KUKA KRL program: ps_stb_geo_c1.src, ps_stb_geo_c1.dat

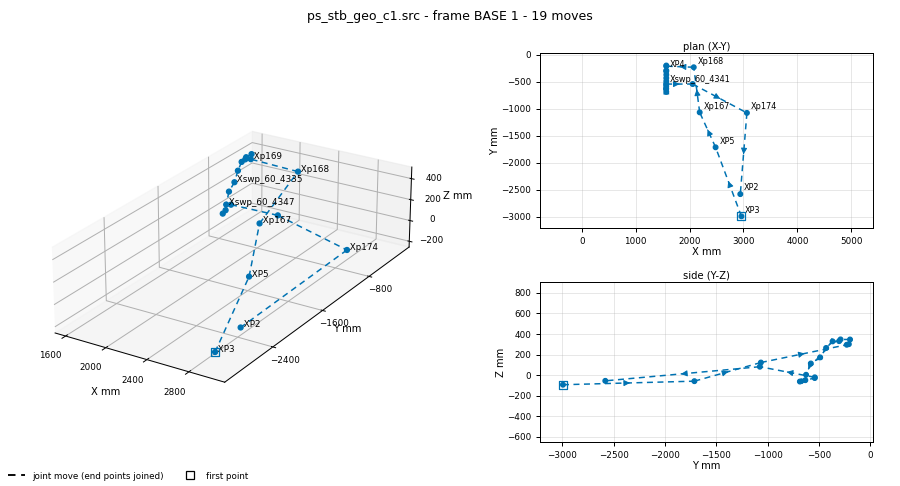
[picture p0: tool path of ps_stb_geo_c1.src in frame BASE 1, 19 of 19 moves have a stored position in this frame; points joined in program order, loops and branches not executed]
--- ps_stb_geo_c1.src ---
&ACCESS RVO
&REL 8
&COMMENT Solda GUN C1 geometria
&PARAM DISKPATH = KRC:\R1\Program
DEF ps_stb_geo_c1( )

;FOLD INI
  ;FOLD BASISTECH INI
    GLOBAL INTERRUPT DECL 3 WHEN $STOPMESS==TRUE DO IR_STOPM ( )
    INTERRUPT ON 3
    BAS (#INITMOV,0 )
  ;ENDFOLD (BASISTECH INI)
;FOLD SPOTTECH INI
USERSPOT(#INIT)
;ENDFOLD (SPOTTECH INI)
;FOLD GRIPPERTECH INI
USER_GRP(0,DUMMY,DUMMY,GDEFAULT)
;ENDFOLD (GRIPPERTECH INI)
  ;FOLD USER INI
    ;Make your modifications here

  ;ENDFOLD (USER INI)
;ENDFOLD (INI)

; Caracterização dos meios de produção:
; Versão Atual:
; 08/06/2013 12:00 Name: P13.050-R1 CHANGES: Solda geometria STB
; Gun C1 (F2 6640 0018 984)

chk_w2_wechs_ok ( )              ; CHECK C1

if MaxStandMenge (1) then
 MaxStandmengeErreicht (1)
endif

IF (NOT(GHOST())) THEN
if Elektrodenwechsel (1) then
 e_fraes2 ()
endif
ENDIF

;FOLD PTP P3 CONT Vel=100 % P_OLP23 Tool[2]:GUN C1 Base[1]:Actros;%{PE}%R 8.2.20,%MKUKATPBASIS,%CMOVE,%VPTP,%P 1:PTP, 2:P3, 3:C_DIS, 5:100, 7:P_OLP23
$BWDSTART=FALSE
PDAT_ACT=PP_OLP23
FDAT_ACT=FP3
BAS(#PTP_PARAMS,100)
PTP XP3 C_DIS
;ENDFOLD
;FOLD PTP P5 CONT Vel=100 % P_OLP24 Tool[2]:GUN C1 Base[1]:Actros;%{PE}%R 8.2.20,%MKUKATPBASIS,%CMOVE,%VPTP,%P 1:PTP, 2:P5, 3:C_DIS, 5:100, 7:P_OLP24
$BWDSTART=FALSE
PDAT_ACT=PP_OLP24
FDAT_ACT=FP5
BAS(#PTP_PARAMS,100)
PTP XP5 C_DIS
;ENDFOLD

;FOLD OUT 3339 'R1 solicita lib soldar geometria' State=TRUE ;%{PE}%R 8.2.20,%MKUKATPBASIS,%COUT,%VOUTX,%P 2:3339, 3:R1 solicita lib soldar geometria, 5:TRUE, 6:
$OUT[3339]=TRUE
;ENDFOLD
;FOLD WAIT FOR ( IN 3339 'Aguarda lib. Soldar geometria' );%{PE}%R 8.2.20,%MKUKATPBASIS,%CEXT_WAIT_FOR,%VEXT_WAIT_FOR,%P 2:, 4:, 5:$IN, 6:3339, 7:Aguarda lib. Soldar geometria, 9:
WAIT FOR  ( $IN[3339] )
;ENDFOLD
;FOLD OUT 3339 'R1 solicita lib soldar geometria' State=FALSE ;%{PE}%R 8.2.20,%MKUKATPBASIS,%COUT,%VOUTX,%P 2:3339, 3:R1 solicita lib soldar geometria, 5:FALSE, 6:
$OUT[3339]=FALSE
;ENDFOLD
;FOLD OUT 3344 'R1 entregou peça geo box' State=FALSE ;%{PE}%R 8.2.20,%MKUKATPBASIS,%COUT,%VOUTX,%P 2:3344, 3:R1 entregou peça geo box, 5:FALSE, 6:
$OUT[3344]=FALSE
;ENDFOLD
;FOLD OUT 3348 'Fora area GEOBOX' State=FALSE ;%{PE}%R 8.2.20,%MKUKATPBASIS,%COUT,%VOUTX,%P 2:3348, 3:Fora area GEOBOX, 5:FALSE, 6:
$OUT[3348]=FALSE
;ENDFOLD

;FOLD PTP p167 CONT Vel=100 % P_OLP6 Tool[2]:GUN C1 Base[1]:Actros;%{PE}%R8.2,%MKUKATPBASIS,%CMOVE,%VPTP,%P 1:PTP, 2:p167, 3:C_DIS, 5:100, 7:P_OLP6
$BWDSTART = FALSE
PDAT_ACT= PP_OLP6
FDAT_ACT= Fp167
BAS(#PTP_PARAMS,100)
PTP Xp167 C_DIS
;ENDFOLD

;FOLD Collision.Monitoring_2_On ;%{PE}%MKUKATPUSER
COLLSTOP( 2, 1 ) ;Interrupt-Controlled
;ENDFOLD

;FOLD PTP p168 CONT Vel=100 % P_OLP7 Tool[2]:GUN C1 Base[1]:Actros;%{PE}%R8.2,%MKUKATPBASIS,%CMOVE,%VPTP,%P 1:PTP, 2:p168, 3:C_DIS, 5:100, 7:P_OLP7
$BWDSTART = FALSE
PDAT_ACT= PP_OLP7
FDAT_ACT= Fp168
BAS(#PTP_PARAMS,100)
PTP Xp168 C_DIS
;ENDFOLD
;FOLD PTP p169 CONT Vel=100 % P_OLP8 Tool[2]:GUN C1 Base[1]:Actros;%{PE}%R8.2,%MKUKATPBASIS,%CMOVE,%VPTP,%P 1:PTP, 2:p169, 3:C_DIS, 5:100, 7:P_OLP8
$BWDSTART = FALSE
PDAT_ACT= PP_OLP8
FDAT_ACT= Fp169
BAS(#PTP_PARAMS,100)
PTP Xp169 C_DIS
;ENDFOLD

;FOLD ; swp_60_4311;%{PE}%R 8.2.20,%MKUKATPBASIS,%CCOMMENT,%VNORMAL,%P 2:swp_60_4311
;ENDFOLD
;FOLD PTP swp_60_4311 P_OLP9 SPOT Gun=1 RETR CLS PgNo1=38 ACTIVE=1 Tool[2]:GUN C1 Base[1]:Actros;%{PE}%R 8.2.2,%MKUKATPSPOT,%CSPOT,%VPTP,%P 1:PTP, 2:swp_60_4311, 3:, 5:100, 7:P_OLP9, 10:1, 12:#FIRST, 14:#CLO, 16:38, 18:1, 20:1, 22:0, 24:1, 25:S_OLP1
$BWDSTART=FALSE
PDAT_ACT=PP_OLP9
FDAT_ACT=Fswp_60_4311
BAS(#PTP_PARAMS,PP_OLP9.VEL)
S_ACT.GUN=1
S_ACT.PAIR=SDEFAULT.PAIR
S_ACT.RETR=#CLO
S_ACT.CLO_TM=1
S_ACT.PGNO1=38
S_ACT.PGNO2=SDEFAULT.PGNO2
S_ACT.PRESS1=SDEFAULT.PRESS1
S_ACT.PRESS2=SDEFAULT.PRESS2
S_READY=FALSE
PTP Xswp_60_4311
USERSPOT(#SPOT, S_ACT)
WAIT FOR S_READY
;ENDFOLD

;FOLD ; swp_60_4317;%{PE}%R 8.2.20,%MKUKATPBASIS,%CCOMMENT,%VNORMAL,%P 2:swp_60_4317
;ENDFOLD
;FOLD PTP swp_60_4317 P_OLP10 SPOT Gun=1 RETR CLS PgNo1=39 ACTIVE=1 Tool[2]:GUN C1 Base[1]:Actros;%{PE}%R 8.2.2,%MKUKATPSPOT,%CSPOT,%VPTP,%P 1:PTP, 2:swp_60_4317, 3:, 5:100, 7:P_OLP10, 10:1, 12:#FIRST, 14:#CLO, 16:39, 18:1, 20:1, 22:0, 24:1, 25:S_OLP2
$BWDSTART=FALSE
PDAT_ACT=PP_OLP10
FDAT_ACT=Fswp_60_4317
BAS(#PTP_PARAMS,PP_OLP10.VEL)
S_ACT.GUN=1
S_ACT.PAIR=SDEFAULT.PAIR
S_ACT.RETR=#CLO
S_ACT.CLO_TM=1
S_ACT.PGNO1=39
S_ACT.PGNO2=SDEFAULT.PGNO2
S_ACT.PRESS1=SDEFAULT.PRESS1
S_ACT.PRESS2=SDEFAULT.PRESS2
S_READY=FALSE
PTP Xswp_60_4317
USERSPOT(#SPOT, S_ACT)
WAIT FOR S_READY
;ENDFOLD

;FOLD PTP P4 CONT Vel=100 % PDAT3 Tool[2]:GUN C1 Base[1]:Actros;%{PE}%R 8.2.20,%MKUKATPBASIS,%CMOVE,%VPTP,%P 1:PTP, 2:P4, 3:C_DIS, 5:100, 7:PDAT3
$BWDSTART=FALSE
PDAT_ACT=PPDAT3
FDAT_ACT=FP4
BAS(#PTP_PARAMS,100)
PTP XP4 C_DIS
;ENDFOLD

;FOLD ; swp_60_4323;%{PE}%R 8.2.20,%MKUKATPBASIS,%CCOMMENT,%VNORMAL,%P 2:swp_60_4323
;ENDFOLD
;FOLD PTP swp_60_4323 P_OLP11 SPOT Gun=1 RETR CLS PgNo1=40 ACTIVE=1 Tool[2]:GUN C1 Base[1]:Actros;%{PE}%R 8.2.2,%MKUKATPSPOT,%CSPOT,%VPTP,%P 1:PTP, 2:swp_60_4323, 3:, 5:100, 7:P_OLP11, 10:1, 12:#FIRST, 14:#CLO, 16:40, 18:1, 20:1, 22:0, 24:1, 25:S_OLP3
$BWDSTART=FALSE
PDAT_ACT=PP_OLP11
FDAT_ACT=Fswp_60_4323
BAS(#PTP_PARAMS,PP_OLP11.VEL)
S_ACT.GUN=1
S_ACT.PAIR=SDEFAULT.PAIR
S_ACT.RETR=#CLO
S_ACT.CLO_TM=1
S_ACT.PGNO1=40
S_ACT.PGNO2=SDEFAULT.PGNO2
S_ACT.PRESS1=SDEFAULT.PRESS1
S_ACT.PRESS2=SDEFAULT.PRESS2
S_READY=FALSE
PTP Xswp_60_4323
USERSPOT(#SPOT, S_ACT)
WAIT FOR S_READY
;ENDFOLD

;FOLD ; swp_60_4329;%{PE}%R 8.2.20,%MKUKATPBASIS,%CCOMMENT,%VNORMAL,%P 2:swp_60_4329
;ENDFOLD
;FOLD PTP swp_60_4329 P_OLP12 SPOT Gun=1 RETR CLS PgNo1=41 ACTIVE=1 Tool[2]:GUN C1 Base[1]:Actros;%{PE}%R 8.2.2,%MKUKATPSPOT,%CSPOT,%VPTP,%P 1:PTP, 2:swp_60_4329, 3:, 5:100, 7:P_OLP12, 10:1, 12:#FIRST, 14:#CLO, 16:41, 18:1, 20:1, 22:0, 24:1, 25:S_OLP4
$BWDSTART=FALSE
PDAT_ACT=PP_OLP12
FDAT_ACT=Fswp_60_4329
BAS(#PTP_PARAMS,PP_OLP12.VEL)
S_ACT.GUN=1
S_ACT.PAIR=SDEFAULT.PAIR
S_ACT.RETR=#CLO
S_ACT.CLO_TM=1
S_ACT.PGNO1=41
S_ACT.PGNO2=SDEFAULT.PGNO2
S_ACT.PRESS1=SDEFAULT.PRESS1
S_ACT.PRESS2=SDEFAULT.PRESS2
S_READY=FALSE
PTP Xswp_60_4329
USERSPOT(#SPOT, S_ACT)
WAIT FOR S_READY
;ENDFOLD

;FOLD ; swp_60_4335;%{PE}%R 8.2.20,%MKUKATPBASIS,%CCOMMENT,%VNORMAL,%P 2:swp_60_4335
;ENDFOLD
;FOLD PTP swp_60_4335 P_OLP13 SPOT Gun=1 RETR CLS PgNo1=42 ACTIVE=1 Tool[2]:GUN C1 Base[1]:Actros;%{PE}%R 8.2.2,%MKUKATPSPOT,%CSPOT,%VPTP,%P 1:PTP, 2:swp_60_4335, 3:, 5:100, 7:P_OLP13, 10:1, 12:#FIRST, 14:#CLO, 16:42, 18:1, 20:1, 22:0, 24:1, 25:S_OLP5
$BWDSTART=FALSE
PDAT_ACT=PP_OLP13
FDAT_ACT=Fswp_60_4335
BAS(#PTP_PARAMS,PP_OLP13.VEL)
S_ACT.GUN=1
S_ACT.PAIR=SDEFAULT.PAIR
S_ACT.RETR=#CLO
S_ACT.CLO_TM=1
S_ACT.PGNO1=42
S_ACT.PGNO2=SDEFAULT.PGNO2
S_ACT.PRESS1=SDEFAULT.PRESS1
S_ACT.PRESS2=SDEFAULT.PRESS2
S_READY=FALSE
PTP Xswp_60_4335
USERSPOT(#SPOT, S_ACT)
WAIT FOR S_READY
;ENDFOLD

;FOLD ; swp_60_4341;%{PE}%R 8.2.20,%MKUKATPBASIS,%CCOMMENT,%VNORMAL,%P 2:swp_60_4341
;ENDFOLD
;FOLD PTP swp_60_4341 P_OLP14 SPOT Gun=1 RETR CLS PgNo1=43 ACTIVE=1 Tool[2]:GUN C1 Base[1]:Actros;%{PE}%R 8.2.2,%MKUKATPSPOT,%CSPOT,%VPTP,%P 1:PTP, 2:swp_60_4341, 3:, 5:100, 7:P_OLP14, 10:1, 12:#FIRST, 14:#CLO, 16:43, 18:1, 20:1, 22:0, 24:1, 25:S_OLP6
$BWDSTART=FALSE
PDAT_ACT=PP_OLP14
FDAT_ACT=Fswp_60_4341
BAS(#PTP_PARAMS,PP_OLP14.VEL)
S_ACT.GUN=1
S_ACT.PAIR=SDEFAULT.PAIR
S_ACT.RETR=#CLO
S_ACT.CLO_TM=1
S_ACT.PGNO1=43
S_ACT.PGNO2=SDEFAULT.PGNO2
S_ACT.PRESS1=SDEFAULT.PRESS1
S_ACT.PRESS2=SDEFAULT.PRESS2
S_READY=FALSE
PTP Xswp_60_4341
USERSPOT(#SPOT, S_ACT)
WAIT FOR S_READY
;ENDFOLD

;FOLD ; swp_60_4347;%{PE}%R 8.2.20,%MKUKATPBASIS,%CCOMMENT,%VNORMAL,%P 2:swp_60_4347
;ENDFOLD
;FOLD PTP swp_60_4347 P_OLP15 SPOT Gun=1 RETR CLS PgNo1=44 ACTIVE=1 Tool[2]:GUN C1 Base[1]:Actros;%{PE}%R 8.2.2,%MKUKATPSPOT,%CSPOT,%VPTP,%P 1:PTP, 2:swp_60_4347, 3:, 5:100, 7:P_OLP15, 10:1, 12:#FIRST, 14:#CLO, 16:44, 18:1, 20:1, 22:0, 24:1, 25:S_OLP7
$BWDSTART=FALSE
PDAT_ACT=PP_OLP15
FDAT_ACT=Fswp_60_4347
BAS(#PTP_PARAMS,PP_OLP15.VEL)
S_ACT.GUN=1
S_ACT.PAIR=SDEFAULT.PAIR
S_ACT.RETR=#CLO
S_ACT.CLO_TM=1
S_ACT.PGNO1=44
S_ACT.PGNO2=SDEFAULT.PGNO2
S_ACT.PRESS1=SDEFAULT.PRESS1
S_ACT.PRESS2=SDEFAULT.PRESS2
S_READY=FALSE
PTP Xswp_60_4347
USERSPOT(#SPOT, S_ACT)
WAIT FOR S_READY
;ENDFOLD

;FOLD PTP p170 CONT Vel=100 % P_OLP16 Tool[2]:GUN C1 Base[1]:Actros;%{PE}%R 8.2.20,%MKUKATPBASIS,%CMOVE,%VPTP,%P 1:PTP, 2:p170, 3:C_DIS, 5:100, 7:P_OLP16
$BWDSTART=FALSE
PDAT_ACT=PP_OLP16
FDAT_ACT=Fp170
BAS(#PTP_PARAMS,100)
PTP Xp170 C_DIS
;ENDFOLD

;FOLD ; swp_60_4353;%{PE}%R 8.2.20,%MKUKATPBASIS,%CCOMMENT,%VNORMAL,%P 2:swp_60_4353
;ENDFOLD
;FOLD PTP swp_60_4353 P_OLP17 SPOT Gun=1 RETR CLS PgNo1=45 ACTIVE=1 Tool[2]:GUN C1 Base[1]:Actros;%{PE}%R 8.2.2,%MKUKATPSPOT,%CSPOT,%VPTP,%P 1:PTP, 2:swp_60_4353, 3:, 5:100, 7:P_OLP17, 10:1, 12:#FIRST, 14:#CLO, 16:45, 18:1, 20:1, 22:0, 24:1, 25:S_OLP8
$BWDSTART=FALSE
PDAT_ACT=PP_OLP17
FDAT_ACT=Fswp_60_4353
BAS(#PTP_PARAMS,PP_OLP17.VEL)
S_ACT.GUN=1
S_ACT.PAIR=SDEFAULT.PAIR
S_ACT.RETR=#CLO
S_ACT.CLO_TM=1
S_ACT.PGNO1=45
S_ACT.PGNO2=SDEFAULT.PGNO2
S_ACT.PRESS1=SDEFAULT.PRESS1
S_ACT.PRESS2=SDEFAULT.PRESS2
S_READY=FALSE
PTP Xswp_60_4353
USERSPOT(#SPOT, S_ACT)
WAIT FOR S_READY
;ENDFOLD

;FOLD PTP P1 CONT Vel=100 % PDAT1 Tool[2]:GUN C1 Base[1]:Actros;%{PE}%R 8.2.20,%MKUKATPBASIS,%CMOVE,%VPTP,%P 1:PTP, 2:P1, 3:C_DIS, 5:100, 7:PDAT1
$BWDSTART=FALSE
PDAT_ACT=PPDAT1
FDAT_ACT=FP1
BAS(#PTP_PARAMS,100)
PTP XP1 C_DIS
;ENDFOLD
;FOLD PTP p171 CONT Vel=100 % P_OLP18 Tool[2]:GUN C1 Base[1]:Actros;%{PE}%R8.2,%MKUKATPBASIS,%CMOVE,%VPTP,%P 1:PTP, 2:p171, 3:C_DIS, 5:100, 7:P_OLP18
$BWDSTART = FALSE
PDAT_ACT= PP_OLP18
FDAT_ACT= Fp171
BAS(#PTP_PARAMS,100)
PTP Xp171 C_DIS
;ENDFOLD
;FOLD PTP p174 CONT Vel=100 % P_OLP21 Tool[2]:GUN C1 Base[1]:Actros;%{PE}%R8.2,%MKUKATPBASIS,%CMOVE,%VPTP,%P 1:PTP, 2:p174, 3:C_DIS, 5:100, 7:P_OLP21
$BWDSTART = FALSE
PDAT_ACT= PP_OLP21
FDAT_ACT= Fp174
BAS(#PTP_PARAMS,100)
PTP Xp174 C_DIS
;ENDFOLD

;FOLD Collision.Monitoring_2_Off . ;%{PE}%MKUKATPUSER
COLLSTOP( 2, 2+0 )
;ENDFOLD
;FOLD OUT 3348 'Fora area GEOBOX' State=TRUE ;%{PE}%R 8.2.20,%MKUKATPBASIS,%COUT,%VOUTX,%P 2:3348, 3:Fora area GEOBOX, 5:TRUE, 6:
$OUT[3348]=TRUE
;ENDFOLD

;FOLD PTP P2 CONT Vel=100 % PDAT2 Tool[2]:GUN C1 Base[1]:Actros;%{PE}%R 8.2.20,%MKUKATPBASIS,%CMOVE,%VPTP,%P 1:PTP, 2:P2, 3:C_DIS, 5:100, 7:PDAT2
$BWDSTART=FALSE
PDAT_ACT=PPDAT2
FDAT_ACT=FP2
BAS(#PTP_PARAMS,100)
PTP XP2 C_DIS
;ENDFOLD

IF (NOT(GHOST())) THEN
if FraesAnf (1) then
 f_fraes2 ()
endif
ENDIF
END

--- ps_stb_geo_c1.dat ---
&ACCESS RVO
&REL 8
&COMMENT Solda GUN C1 geometria
&PARAM DISKPATH = KRC:\R1\Program
DEFDAT ps_stb_geo_c1
;FOLD EXTERNAL DECLARATIONS;%{PE}%MKUKATPBASIS,%CEXT,%VCOMMON,%P
;FOLD GRIPPERTECH EXT
EXT  H50 (INT  :IN,INT  :IN,INT  :IN,GRP_TYP  :IN )
;ENDFOLD (GRIPPERTECH EXT)
;FOLD SPOTTECH EXT
EXT  USERSPOT (S_COMMAND  :IN,SPOT_TYPE  :IN )
;ENDFOLD (SPOTTECH EXT)
;FOLD BASISTECH EXT;%{PE}%MKUKATPBASIS,%CEXT,%VEXT,%P
EXT  BAS (BAS_COMMAND  :IN,REAL  :IN )
DECL INT SUCCESS
;ENDFOLD (BASISTECH EXT)
;FOLD USER EXT;%{E}%MKUKATPUSER,%CEXT,%VEXT,%P
;Make your modifications here

;ENDFOLD (USER EXT)
;ENDFOLD (EXTERNAL DECLARATIONS)

;# ============ START PATH : swp_p13050r1_stb_geo_c1 =============
DECL FDAT Fp167={TOOL_NO 2,BASE_NO 1,IPO_FRAME #BASE,POINT2[] " "}
DECL PDAT PP_OLP6={VEL 100.0,ACC 100.0,APO_DIST 100.0,APO_MODE #CDIS}
DECL E6POS Xp167={X 2187.70288,Y -1065.02905,Z 122.171501,A 154.582001,B -61.0634308,C 20.8292103,S 2,T 42,E1 -4705.90723,E2 0.0,E3 0.0,E4 0.0,E5 0.0,E6 0.0}
DECL FDAT Fp168={TOOL_NO 2,BASE_NO 1,IPO_FRAME #BASE,POINT2[] " "}
DECL PDAT PP_OLP7={VEL 100.0,ACC 100.0,APO_DIST 100.0,APO_MODE #CDIS}
DECL E6POS Xp168={X 2077.50098,Y -228.445694,Z 295.414093,A 74.1307068,B -87.3236465,C 85.4994583,S 2,T 42,E1 -5004.70117,E2 0.0,E3 0.0,E4 0.0,E5 0.0,E6 0.0}
DECL FDAT Fp169={TOOL_NO 2,BASE_NO 1,IPO_FRAME #BASE,POINT2[] " "}
DECL PDAT PP_OLP8={VEL 100.0,ACC 100.0,APO_DIST 100.0,APO_MODE #CDIS}
DECL E6POS Xp169={X 1568.01196,Y -208.078003,Z 301.009186,A 0.0,B -90.0004272,C 179.999802,S 2,T 42,E1 -5004.70215,E2 0.0,E3 0.0,E4 0.0,E5 0.0,E6 0.0}
DECL FDAT Fswp_60_4311={TOOL_NO 2,BASE_NO 1,IPO_FRAME #BASE,POINT2[] " "}
DECL PDAT PP_OLP9={VEL 100.0,ACC 100.0,APO_DIST 0.0}
DECL SPOT_TYPE SS_OLP1={GUN 1,PAIR #FIRST,RETR #CLO,CLO_TM 0,PGNO1 1,PRESS1 1.0,PGNO2 0,PRESS2 0.0}
DECL E6POS Xswp_60_4311={X 1568.65002,Y -196.404297,Z 346.485199,A -89.9976273,B -74.8812866,C -90.0025864,S 2,T 42,E1 -5004.71094,E2 0.0,E3 0.0,E4 0.0,E5 0.0,E6 0.0}
DECL FDAT Fswp_60_4317={TOOL_NO 2,BASE_NO 1,IPO_FRAME #BASE,POINT2[] " "}
DECL PDAT PP_OLP10={VEL 100.0,ACC 100.0,APO_DIST 0.0}
DECL SPOT_TYPE SS_OLP2={GUN 1,PAIR #FIRST,RETR #CLO,CLO_TM 0,PGNO1 1,PRESS1 1.0,PGNO2 0,PRESS2 0.0}
DECL E6POS Xswp_60_4317={X 1568.66296,Y -288.891296,Z 347.407715,A -90.0009689,B -74.8817062,C -89.9984818,S 2,T 42,E1 -5004.7041,E2 0.0,E3 0.0,E4 0.0,E5 0.0,E6 0.0}
DECL FDAT Fswp_60_4323={TOOL_NO 2,BASE_NO 1,IPO_FRAME #BASE,POINT2[] " "}
DECL PDAT PP_OLP11={VEL 100.0,ACC 100.0,APO_DIST 0.0}
DECL SPOT_TYPE SS_OLP3={GUN 1,PAIR #FIRST,RETR #CLO,CLO_TM 0,PGNO1 1,PRESS1 1.0,PGNO2 0,PRESS2 0.0}
DECL E6POS Xswp_60_4323={X 1568.86304,Y -366.544891,Z 328.342194,A -90.0,B -55.9611206,C -90.0,S 2,T 42,E1 -5004.70117,E2 0.0,E3 0.0,E4 0.0,E5 0.0,E6 0.0}
DECL FDAT Fswp_60_4329={TOOL_NO 2,BASE_NO 1,IPO_FRAME #BASE,POINT2[] " "}
DECL PDAT PP_OLP12={VEL 100.0,ACC 100.0,APO_DIST 0.0}
DECL SPOT_TYPE SS_OLP4={GUN 1,PAIR #FIRST,RETR #CLO,CLO_TM 0,PGNO1 1,PRESS1 1.0,PGNO2 0,PRESS2 0.0}
DECL E6POS Xswp_60_4329={X 1568.06799,Y -428.806396,Z 264.020203,A -90.0036011,B -42.844841,C -89.9937363,S 2,T 10,E1 -5004.70313,E2 0.0,E3 0.0,E4 0.0,E5 0.0,E6 0.0}
DECL FDAT Fswp_60_4335={TOOL_NO 2,BASE_NO 1,IPO_FRAME #BASE,POINT2[] " "}
DECL PDAT PP_OLP13={VEL 100.0,ACC 100.0,APO_DIST 0.0}
DECL SPOT_TYPE SS_OLP5={GUN 1,PAIR #FIRST,RETR #CLO,CLO_TM 0,PGNO1 1,PRESS1 1.0,PGNO2 0,PRESS2 0.0}
DECL E6POS Xswp_60_4335={X 1568.06799,Y -487.247894,Z 172.195496,A -89.9989166,B -48.9620399,C -90.0007324,S 2,T 10,E1 -5004.70117,E2 0.0,E3 0.0,E4 0.0,E5 0.0,E6 0.0}
DECL FDAT Fswp_60_4341={TOOL_NO 2,BASE_NO 1,IPO_FRAME #BASE,POINT2[] " "}
DECL PDAT PP_OLP14={VEL 100.0,ACC 100.0,APO_DIST 0.0}
DECL SPOT_TYPE SS_OLP6={GUN 1,PAIR #FIRST,RETR #CLO,CLO_TM 0,PGNO1 1,PRESS1 1.0,PGNO2 0,PRESS2 0.0}
DECL E6POS Xswp_60_4341={X 1567.16101,Y -578.509216,Z 112.906197,A -90.0000229,B -38.1195297,C -89.9997635,S 2,T 10,E1 -5004.70215,E2 0.0,E3 0.0,E4 0.0,E5 0.0,E6 0.0}
DECL FDAT Fswp_60_4347={TOOL_NO 2,BASE_NO 1,IPO_FRAME #BASE,POINT2[] " "}
DECL PDAT PP_OLP15={VEL 100.0,ACC 100.0,APO_DIST 0.0}
DECL SPOT_TYPE SS_OLP7={GUN 1,PAIR #FIRST,RETR #CLO,CLO_TM 0,PGNO1 1,PRESS1 1.0,PGNO2 0,PRESS2 0.0}
DECL E6POS Xswp_60_4347={X 1566.90295,Y -624.828796,Z 2.8932569,A -89.9996338,B -8.81437397,C -90.000412,S 2,T 10,E1 -5004.70313,E2 0.0,E3 0.0,E4 0.0,E5 0.0,E6 0.0}
DECL FDAT Fp170={TOOL_NO 2,BASE_NO 1,IPO_FRAME #BASE,POINT2[] " ",TQ_STATE FALSE}
DECL PDAT PP_OLP16={VEL 100.0,ACC 100.0,APO_DIST 100.0,APO_MODE #CDIS}
DECL E6POS Xp170={X 1564.73401,Y -631.993408,Z -49.9609299,A -90.0104828,B 9.44801426,C -89.0347672,S 2,T 10,E1 -5004.70117,E2 0.0,E3 0.0,E4 0.0,E5 0.0,E6 0.0}
DECL FDAT Fswp_60_4353={TOOL_NO 2,BASE_NO 1,IPO_FRAME #BASE,POINT2[] " "}
DECL PDAT PP_OLP17={VEL 100.0,ACC 100.0,APO_DIST 0.0}
DECL SPOT_TYPE SS_OLP8={GUN 1,PAIR #FIRST,RETR #CLO,CLO_TM 0,PGNO1 1,PRESS1 1.0,PGNO2 0,PRESS2 0.0}
DECL E6POS Xswp_60_4353={X 1568.02905,Y -685.09967,Z -63.1332512,A -90.0916519,B 11.0299101,C -89.0324097,S 2,T 10,E1 -5004.66895,E2 0.0,E3 0.0,E4 0.0,E5 0.0,E6 0.0}
DECL FDAT Fp171={TOOL_NO 2,BASE_NO 1,IPO_FRAME #BASE,POINT2[] " "}
DECL PDAT PP_OLP18={VEL 100.0,ACC 100.0,APO_DIST 100.0,APO_MODE #CDIS}
DECL E6POS Xp171={X 2057.34399,Y -539.947327,Z -21.8766994,A -85.5985489,B 8.36809731,C -61.0904999,S 2,T 10,E1 -5004.70117,E2 0.0,E3 0.0,E4 0.0,E5 0.0,E6 0.0}
DECL FDAT Fp174={TOOL_NO 2,BASE_NO 1,IPO_FRAME #BASE,POINT2[] " "}
DECL PDAT PP_OLP21={VEL 100.0,ACC 100.0,APO_DIST 100.0,APO_MODE #CDIS}
DECL E6POS Xp174={X 3063.42212,Y -1075.047,Z 81.3437271,A -97.5164337,B 21.5872192,C -13.7264299,S 2,T 10,E1 -4617.95508,E2 0.0,E3 0.0,E4 0.0,E5 0.0,E6 0.0}
DECL BASIS_SUGG_T LAST_BASIS={POINT1[] "P7                      ",POINT2[] "P7                      ",CP_PARAMS[] "CPDAT0                  ",PTP_PARAMS[] "PDAT5                   ",CONT[] "                        ",CP_VEL[] "2.0                     ",PTP_VEL[] "100                     ",SYNC_PARAMS[] "SYNCDAT                 ",SPL_NAME[] "S0                      "}
DECL E6POS XP1={X 1564.65295,Y -540.241882,Z -28.7788105,A -90.0104828,B 9.44801426,C -89.0347672,S 2,T 10,E1 -5004.70117,E2 0.0,E3 0.0,E4 0.0,E5 0.0,E6 0.0}
DECL FDAT FP1={TOOL_NO 2,BASE_NO 1,IPO_FRAME #BASE,POINT2[] " ",TQ_STATE FALSE}
DECL PDAT PPDAT1={VEL 100.0,ACC 100.0,APO_DIST 100.0,APO_MODE #CDIS}
DECL E6POS XP2={X 2940.87305,Y -2581.30591,Z -56.23843,A -12.3740101,B 2.19144797,C 0.804901302,S 2,T 2,E1 -4016.84912,E2 0.0,E3 0.0,E4 0.0,E5 0.0,E6 0.0}
DECL FDAT FP2={TOOL_NO 2,BASE_NO 1,IPO_FRAME #BASE,POINT2[] " ",TQ_STATE FALSE}
DECL PDAT PPDAT2={VEL 100.0,ACC 100.0,APO_DIST 0.0,APO_MODE #CDIS}
DECL SPOT_SUGG_T LAST_SPOT={GUN[] "1                       ",RETR_CMD[] "#OPN                    ",CHOISE[] "#FIRST                  ",CLO_TM[] "0                       ",PGNO1[] "1                       ",PRESS1[] "0                       ",PGNO2[] "1                       ",PRESS2[] "0                       ",SPOT_PARAMS[] "NORMAL                  "}
DECL PDAT PP_OLP23={VEL 100.0,ACC 100.0,APO_DIST 0.0,APO_MODE #CDIS}
DECL E6POS XP3={X 2961.71509,Y -2993.75195,Z -94.1015167,A -120.318604,B -15.7421103,C -6.4170928,S 2,T 42,E1 -3538.53101,E2 0.0,E3 0.0,E4 0.0,E5 0.0,E6 0.0}
DECL FDAT FP3={TOOL_NO 2,BASE_NO 1,IPO_FRAME #BASE,POINT2[] " "}
DECL E6POS XP4={X 1567.18396,Y -302.475586,Z 330.597412,A -90.0009079,B -74.8817062,C -89.9986877,S 2,T 42,E1 -5004.70508,E2 0.0,E3 0.0,E4 0.0,E5 0.0,E6 0.0}
DECL FDAT FP4={TOOL_NO 2,BASE_NO 1,IPO_FRAME #BASE,POINT2[] " ",TQ_STATE FALSE}
DECL PDAT PPDAT3={VEL 100.0,ACC 100.0,APO_DIST 100.0,APO_MODE #CDIS}
DECL PDAT PP_OLP24={VEL 100.0,ACC 100.0,APO_DIST 100.0,APO_MODE #CDIS}
DECL E6POS XP5={X 2482.64209,Y -1713.11694,Z -59.4795418,A 169.485504,B -20.3076706,C 0.113910303,S 2,T 42,E1 -4233.12207,E2 0.0,E3 0.0,E4 0.0,E5 0.0,E6 0.0}
DECL FDAT FP5={TOOL_NO 2,BASE_NO 1,IPO_FRAME #BASE,POINT2[] " "}
ENDDAT
